FUNCTION FgenerateRandom : Lreal // := rawValue + rawValue*percent* random
VAR_INPUT
	percent : LREAL ;// percent of vabration random +percent
	rawValue : LREAL;
	ValueDrandGenerate : LREAL;
END_VAR
VAR_OUTPUT
	
END_VAR
VAR
	
	
END_VAR

FgenerateRandom := rawValue + rawValue * percent * ValueDrandGenerate;

END_FUNCTION

(* stored: Version 1.1.0.1, ProductVersion 3.1.4024.12
   POU FgenerateRandom: Id {f342d321-aaf6-4252-9c7b-055366d9aa56}, SpecialFunc None *)
